Staubli VAL3: FrameItem.pjx

--- FrameItem.pjx ---
Parameters version=s7.6.1 stackSize=5000 millimeterUnit=true
Program file=start.pgx
Program file=stop.pgx
Data file=FrameItem.dtx

--- FrameItem.dtx ---
public frame fFrame = {fatherId=world[0]}
public pointRx pO = {fatherId=world[0]}
public pointRx pX = {fatherId=world[0]}
public pointRx pY = {fatherId=world[0]}
public string sName
